// TIA Portal V20 export
TYPE "LER_typeSequenceRelation"
// stored: Access Published
   STRUCT
      preOperationCheck { ExternalWritable := 'False'} : Struct   // Check The Status Of Each Homing
         Bool1 : Bool;
         Bool2 : Bool;
         Bool3 : Bool;
         Bool4 : Bool;
         Bool5 : Bool;
         Bool6 : Bool;
         Bool7 : Bool;
         Bool8 : Bool;
         Bool9 : Bool;
         Bool10 : Bool;
         Bool11 : Bool;
         Bool12 : Bool;
         Bool13 : Bool;
         Bool14 : Bool;
         Bool15 : Bool;
         Bool16 : Bool;
         Bool17 : Bool;
         Bool18 : Bool;
         Bool19 : Bool;
         Bool20 : Bool;
      END_STRUCT;
      selectJobStatus { ExternalWritable := 'False'} : Array[0..39] of "LAF_typeJobStatus";
      jobInterface { ExternalWritable := 'False'} : Array[0..39] of "LER_typeJobInterface";   // Interface To Check Equipment Modules Status
   END_STRUCT;
END_TYPE
